// TIA Portal project "Lavadora" (V14)

(* hardware
DEVICE "S7-1200 station_1"  S7-1200 Station
   slot 0: "Rack_0"  Rack  V1.0
   slot 1: "PLC_1"  CPU 1214C DC/DC/DC  6ES7 214-1AG40-0XB0  V4.2
*)

// ===== PLC "PLC_1"  CPU 1214C DC/DC/DC =====

VAR_GLOBAL   // PLC tag table "Entradas_Analogas"
   "Sensor_Puerta" AT %I0.7 : Bool;
END_VAR

VAR_GLOBAL   // PLC tag table "Entradas_Digitales"
   "Start" AT %I0.0 : Bool;   // 1 presiono - 0 no presiono
   "Pausa" AT %I0.1 : Bool;   // 1 no presiono - 0 presiono
   "Stop" AT %I0.2 : Bool;   // 1 sin presionar - 0 presionado
   "Nivel_Alto" AT %I0.3 : Bool;   // 1 presiono - 0 no presiono
   "Nivel_Medio" AT %I0.4 : Bool;   // 1 presiono - 0 no presiono
   "Nivel_Bajo" AT %I0.5 : Bool;   // 1 presiono - 0 no presiono
   "Nivel_Vacio" AT %I0.6 : Bool;   // 1 presiono - 0 no presiono
END_VAR

DATA_BLOCK "HMI_BD"   // DB1
{ S7_Optimized_Access := 'TRUE' }
VERSION : 0.1
BEGIN
END_DATA_BLOCK

FUNCTION "Alarmas" : Void   // FC1, LAD
{ S7_Optimized_Access := 'TRUE' }
VERSION : 0.1
BEGIN
END_FUNCTION

FUNCTION "VariablesHMI" : Void   // FC2, LAD
{ S7_Optimized_Access := 'TRUE' }
VERSION : 0.1
BEGIN
END_FUNCTION

FUNCTION "Control_Valvulas" : Void   // FC3, LAD
{ S7_Optimized_Access := 'TRUE' }
VERSION : 0.1
BEGIN
END_FUNCTION

FUNCTION "Variador" : Void   // FC4, LAD
{ S7_Optimized_Access := 'TRUE' }
VERSION : 0.1
BEGIN
END_FUNCTION

ORGANIZATION_BLOCK "Main"   // OB1, LAD, ProgramCycle
TITLE = "Main Program Sweep (Cycle)"
{ S7_Optimized_Access := 'TRUE' }
VERSION : 0.1
   VAR_INPUT
      Initial_Call : Bool;   // Initial call of this OB
      Remanence : Bool;   // =True, if remanent data are available
   END_VAR
BEGIN
END_ORGANIZATION_BLOCK